FUNCTION F_CalcTD400Checksum : BYTE
VAR_INPUT
    i_abData: ARRAY[0..23] OF BYTE;
END_VAR
VAR
    bChecksum: BYTE;
    i: INT;
END_VAR

bChecksum := i_abData[0];
FOR i:=1 TO 22 DO
    bChecksum := bChecksum XOR i_abData[i];
END_FOR
F_CalcTD400Checksum := bChecksum;

END_FUNCTION

(* stored: Version 1.1.0.1, ProductVersion 3.1.4024.12
   POU F_CalcTD400Checksum: Id {78a78f8f-5f94-4917-91dd-6746146c5f0e}, SpecialFunc None *)
